// TIA Portal V17 export
// export: Created 2024-08-09T12:53:18.2395984Z, ExportSetting WithDefaults, DisplayName Totally Integrated Automation Portal, DisplayVersion V17 Update 7, DisplayName TIA Portal Openness, DisplayVersion V17 Update 7, DisplayName TIA Portal Version Control Interface, DisplayVersion V17, DisplayName STEP 7 Professional, DisplayVersion V17 Update 7, DisplayName STEP 7 Safety, DisplayVersion V17 Update 6, DisplayName WinCC Professional, DisplayVersion V17 Update 7
TYPE "Vis_Silo"
// stored: IsFailsafeCompliant false
   STRUCT
      _Mobile : Int;
      _Etp : SInt;
      _EtpPrec { ExternalAccessible := 'False'; ExternalVisible := 'False'; ExternalWritable := 'False'} : SInt;
      _Marche : Bool;
      _Nb : Bool;
      _SecPorte : Bool;
   END_STRUCT;
END_TYPE
